Omron Sysmac Studio project SPA_Q10 (Sysmac Studio 1.23.0.14, StandardProject)

# Controller new_Controller_0: NX1P2-1040DT1 version 1.18
Task PrimaryTask (priority 4, period or condition 2000): Programa0

VAR_GLOBAL
    rawKgAcetona : INT;  (* Señal de corriente sensor tanque acetona; at BuiltInIO://opt/#0/Ch1_Analog_Input_Value *)
    PP : BOOL;  (* Pulsador de Paro; at BuiltInIO://cpu/#0/Input_Bit_00 *)
    PM : BOOL;  (* Pulsador de Marcha; at BuiltInIO://cpu/#0/Input_Bit_01 *)
    PR : BOOL;  (* Pulsador de Reset; at BuiltInIO://cpu/#0/Input_Bit_02 *)
    V1 : BOOL;  (* Avance Motor; at BuiltInIO://cpu/#0/Output_Bit_00 *)
    V2 : BOOL;  (* Retroceso Motor; at BuiltInIO://cpu/#0/Output_Bit_01 *)
    V3 : BOOL;  (* Multivelocidad 1; at BuiltInIO://cpu/#0/Output_Bit_02 *)
    V4 : BOOL;  (* Multivelocidad 2; at BuiltInIO://cpu/#0/Output_Bit_03 *)
    V5 : BOOL;  (* Multivelocidad 3; at BuiltInIO://cpu/#0/Output_Bit_04 *)
    rawKgAcido : INT;  (* Señal de corriente sensor tanque acido nitrico; at BuiltInIO://opt/#0/Ch2_Analog_Input_Value *)
END_VAR
VAR_GLOBAL RETAIN
    AlturaTanque AT %D10 : REAL;  (* published *)
END_VAR

PROGRAM Programa0
VAR
    kgAcetona : REAL;
    volumenAcetona : REAL;
    kgAcetonaReal : REAL;
    EstadoTanque : INT;
END_VAR
VAR_EXTERNAL
    V1 : BOOL;
    rawKgAcetona : INT;
    AlturaTanque : REAL;
END_VAR

(* Section Calculos: ladder, written here as Structured Text *)

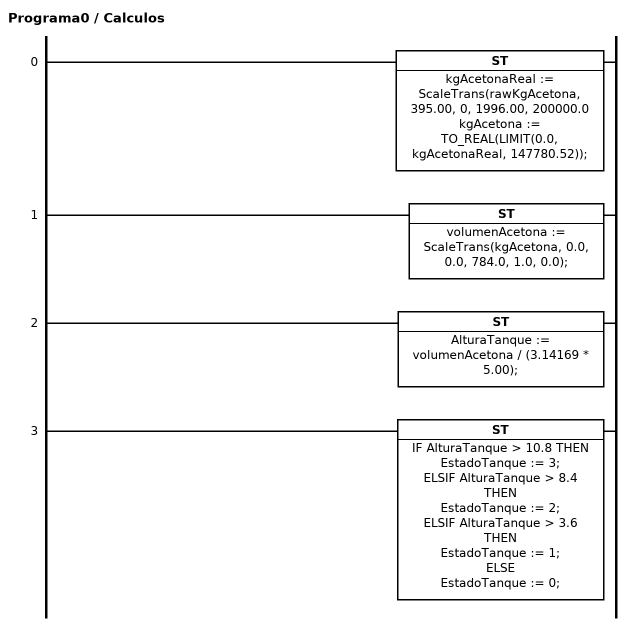
(* Rung 0 *)
kgAcetonaReal := ScaleTrans(rawKgAcetona, 395.00, 0, 1996.00, 200000.00, 0);
kgAcetona := TO_REAL(LIMIT(0.0, kgAcetonaReal, 147780.52));
(* Rung 1 *)
volumenAcetona := ScaleTrans(kgAcetona, 0.0, 0.0, 784.0, 1.0, 0.0);
(* Rung 2 *)
AlturaTanque := volumenAcetona / (3.14169 * 5.00);
(* Rung 3 *)
IF AlturaTanque > 10.8 THEN
	EstadoTanque := 3;
ELSIF AlturaTanque > 8.4 THEN
	EstadoTanque := 2;
ELSIF AlturaTanque > 3.6 THEN
	EstadoTanque := 1;
ELSE
	EstadoTanque := 0;
END_PROGRAM